(* Logix 5000 project; controller QA_DC vendor 1 type 14 code 164 rev 32.16; software revision 32.04; part 3 of 3 *)
(* tags used below, declared in another part *)
   LN99_1st_Station_Break_Code : DINT;
   LN99_Break_LineWide : BOOL;
   LN99_FROM_DC1_MAIN_MESSAGES : DINT[20];
   LN99_Schedule : UDT_Current_Status;
   LN99_TO_DC1_MAIN_MESSAGE_D : DINT[10];   // WORK CENTER D CONSUME TAG
   LN99_TO_DC1_MAIN_MESSAGE_E : DINT[10];   // WORK CENTER E CONSUME TAG
   LN99_TO_DC1_SUB_MESSAGE_C : DINT[10];   // WORK CENTER C CONSUME TAG
   LN99_TO_DC1_SUB_MESSAGE_E : DINT[10];   // WORK CENTER E CONSUME TAG
   LN99ECS01 : DINT;   // WORK STATION EAST SIDE WORKCENTER C SUBLINE STATION 01
   LN99ECS02 : DINT;   // WORK STATION EAST SIDE WORKCENTER C SUBLINE STATION 02
   LN99ECS03 : DINT;   // WORK STATION EAST SIDE WORKCENTER C SUBLINE STATION 03
   LN99EES01 : DINT;   // WORK STATION EAST SIDE WORK CENTER E SUBLINE STATION 01
   LN99EES02 : DINT;   // WORK STATION EAST SIDE WORK CENTER E SUBLINE STATION 02
   LN99EES03 : DINT;   // WORK STATION EAST SIDE WORK CENTER E SUBLINE STATION 03
   LN99NDM01 : DINT;   // WORK STATION NORTH SIDE WORKCENTER D MAINLINE STATION 01
   LN99NDM02 : DINT;   // WORK STATION NORTH SIDE WORK CENTER D MAINLINE STATION 02
   LN99NDM03 : DINT;   // WORK STATION NORTH SIDE WORK CENTER D MAINLINE STATION 03
   LN99NDM04 : DINT;   // WORK STATION NORTH SIDE WORK CENTER D MAINLINE STATION 04
   LN99NEM01 : DINT;   // WORK STATION NORTH SIDE WORK CENTER E MAIN LINE STATION 01
   LN99NEM02 : DINT;   // WORK STATION NORTH SIDE WORK CENTER E MAINLINE STATION 02
   LN99NEM03 : DINT;   // WORK STATION NORTH SIDE WORK CENTER E MAINLINE STATION 03
   LN99NEM04 : DINT;   // WORK STATION NORTH SIDE WORK CENTER E MAINLINE STATION 04
   LN99NEM05 : DINT;   // WORK STATION NORTH SIDE WORK CENTER E MAINLINE STATION 05
   LN99SDM01 : DINT;   // WORK STATION SOUTH SIDE WORKCENTER D MAINLINE STATION 01
   LN99SDM02 : DINT;   // WORK STATION SOUTH SIDE WORK CENTER D MAINLINE STATION 02
   LN99SDM03 : DINT;   // WORK STATION SOUTH SIDE WORK CENTER D MAINLINE STATION 03
   LN99SDM04 : DINT;   // WORK STATION SOUTH SIDE WORK CENTER D MAINLINE STATION 04
   LN99SEM01 : DINT;   // WORK STATION SOUTH SIDE WORK CENTER E MAINLINE STATION 01
   LN99SEM02 : DINT;   // WORK STATION SOUTH SIDE WORK CENTER E MAINLINE STATION 02
   LN99SEM04 : DINT;   // WORK STATION SOUTH SIDE WORK CENTER E MAINLINE STATION 04
   LN99SEM05 : DINT;   // WORK STATION SOUTH SIDE WORK CENTER E MAINLINE STATION 05
   LN99WCS01 : DINT;   // WORK STATION WEST SIDE WORKCENTER C SUBLINE STATION 01
   LN99WCS02 : DINT;   // WORK STATION WEST SIDE WORKCENTER C SUBLINE STATION 02
   LN99WCS03 : DINT;   // WORK STATION WEST SIDE WORKCENTER C SUBLINE STATION 03
   LN99WES01 : DINT;   // WORK STATION WEST SIDE WORK CENTER E SUBLINE STATION 01
   LN99WES02 : DINT;   // WORK STATION WEST SIDE WORK CENTER E SUBLINE STATION 02
   LN99WES03 : DINT;   // WORK STATION WEST SIDE WORK CENTER E SUBLINE STATION 03
(* LN99, continued *)

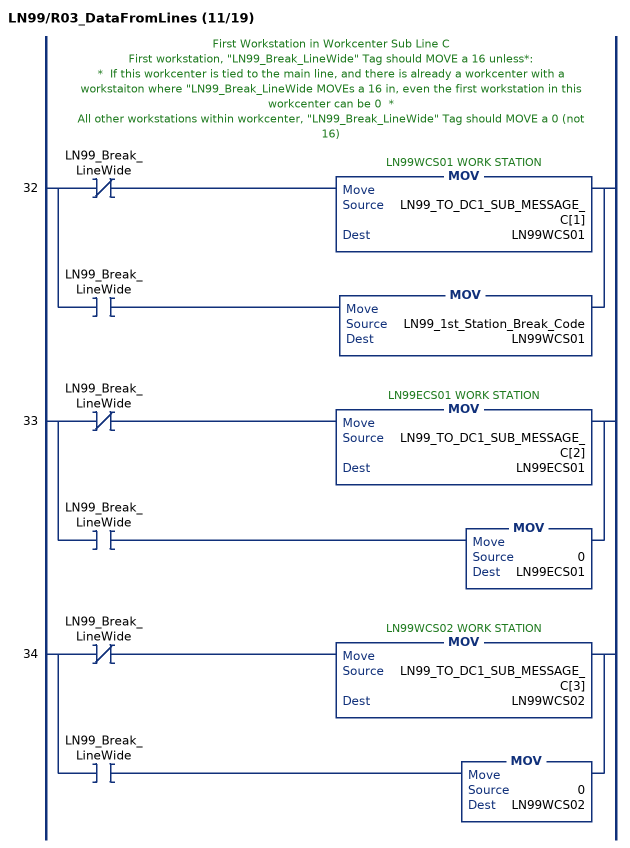
   [picture p52: LN99/R03_DataFromLines rungs 32-34]
   // First Workstation in Workcenter Sub Line C
   // First workstation, "LN99_Break_LineWide" Tag should MOVE a 16 unless*:
   // *  If this workcenter is tied to the main line, and there is already a workcenter with a workstaiton where "LN99_Break_LineWide MOVEs a 16 in, even the first workstation in this workcenter can be 0  *
   // All other workstations within workcenter, "LN99_Break_LineWide" Tag should MOVE a 0 (not 16)
   32: [XIO(LN99_Break_LineWide) MOV(LN99_TO_DC1_SUB_MESSAGE_C[1],LN99WCS01) ,XIC(LN99_Break_LineWide) MOV(LN99_1st_Station_Break_Code,LN99WCS01) ];
   33: [XIO(LN99_Break_LineWide) MOV(LN99_TO_DC1_SUB_MESSAGE_C[2],LN99ECS01) ,XIC(LN99_Break_LineWide) MOV(0,LN99ECS01) ];
   34: [XIO(LN99_Break_LineWide) MOV(LN99_TO_DC1_SUB_MESSAGE_C[3],LN99WCS02) ,XIC(LN99_Break_LineWide) MOV(0,LN99WCS02) ];
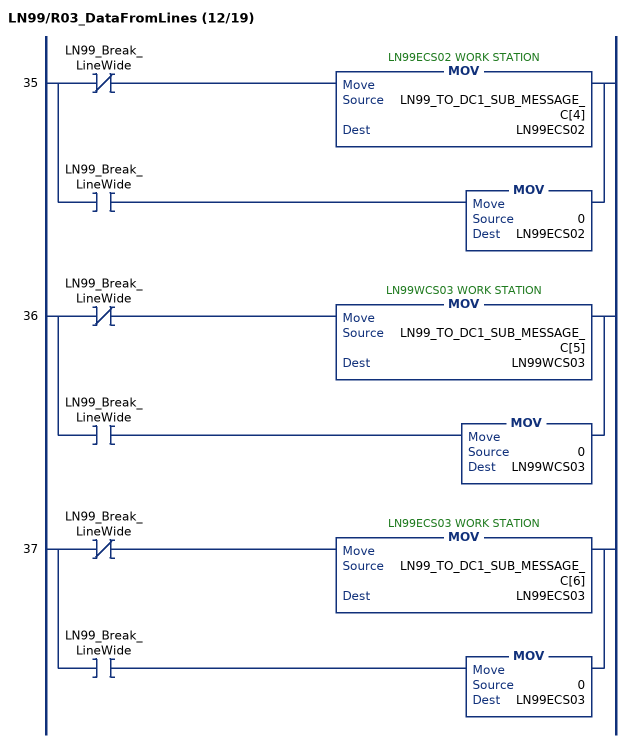
   35: [XIO(LN99_Break_LineWide) MOV(LN99_TO_DC1_SUB_MESSAGE_C[4],LN99ECS02) ,XIC(LN99_Break_LineWide) MOV(0,LN99ECS02) ];
   36: [XIO(LN99_Break_LineWide) MOV(LN99_TO_DC1_SUB_MESSAGE_C[5],LN99WCS03) ,XIC(LN99_Break_LineWide) MOV(0,LN99WCS03) ];
   37: [XIO(LN99_Break_LineWide) MOV(LN99_TO_DC1_SUB_MESSAGE_C[6],LN99ECS03) ,XIC(LN99_Break_LineWide) MOV(0,LN99ECS03) ];
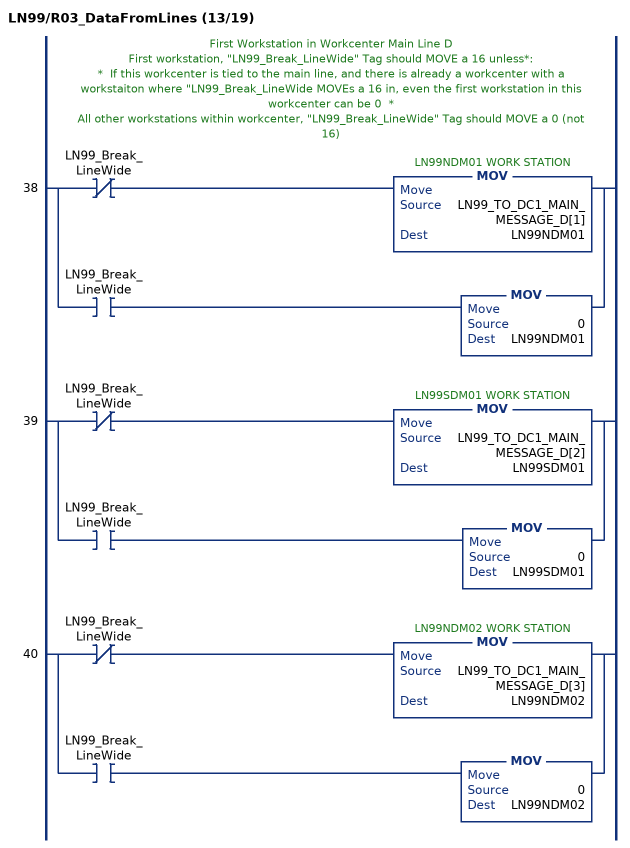
   // First Workstation in Workcenter Main Line D
   // First workstation, "LN99_Break_LineWide" Tag should MOVE a 16 unless*:
   // *  If this workcenter is tied to the main line, and there is already a workcenter with a workstaiton where "LN99_Break_LineWide MOVEs a 16 in, even the first workstation in this workcenter can be 0  *
   // All other workstations within workcenter, "LN99_Break_LineWide" Tag should MOVE a 0 (not 16)
   38: [XIO(LN99_Break_LineWide) MOV(LN99_TO_DC1_MAIN_MESSAGE_D[1],LN99NDM01) ,XIC(LN99_Break_LineWide) MOV(0,LN99NDM01) ];
   39: [XIO(LN99_Break_LineWide) MOV(LN99_TO_DC1_MAIN_MESSAGE_D[2],LN99SDM01) ,XIC(LN99_Break_LineWide) MOV(0,LN99SDM01) ];
   40: [XIO(LN99_Break_LineWide) MOV(LN99_TO_DC1_MAIN_MESSAGE_D[3],LN99NDM02) ,XIC(LN99_Break_LineWide) MOV(0,LN99NDM02) ];
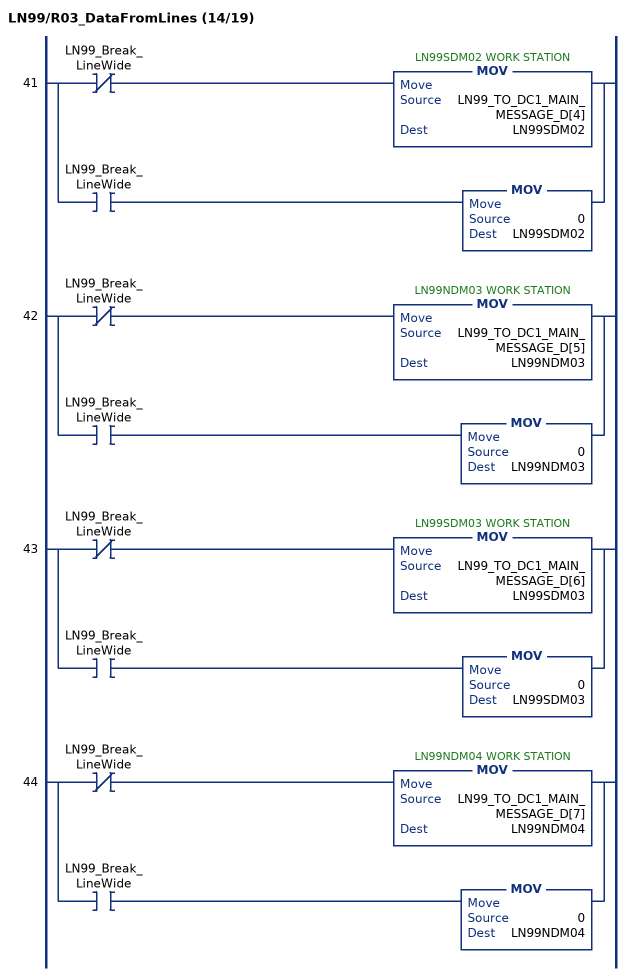
   41: [XIO(LN99_Break_LineWide) MOV(LN99_TO_DC1_MAIN_MESSAGE_D[4],LN99SDM02) ,XIC(LN99_Break_LineWide) MOV(0,LN99SDM02) ];
   42: [XIO(LN99_Break_LineWide) MOV(LN99_TO_DC1_MAIN_MESSAGE_D[5],LN99NDM03) ,XIC(LN99_Break_LineWide) MOV(0,LN99NDM03) ];
   43: [XIO(LN99_Break_LineWide) MOV(LN99_TO_DC1_MAIN_MESSAGE_D[6],LN99SDM03) ,XIC(LN99_Break_LineWide) MOV(0,LN99SDM03) ];
   44: [XIO(LN99_Break_LineWide) MOV(LN99_TO_DC1_MAIN_MESSAGE_D[7],LN99NDM04) ,XIC(LN99_Break_LineWide) MOV(0,LN99NDM04) ];
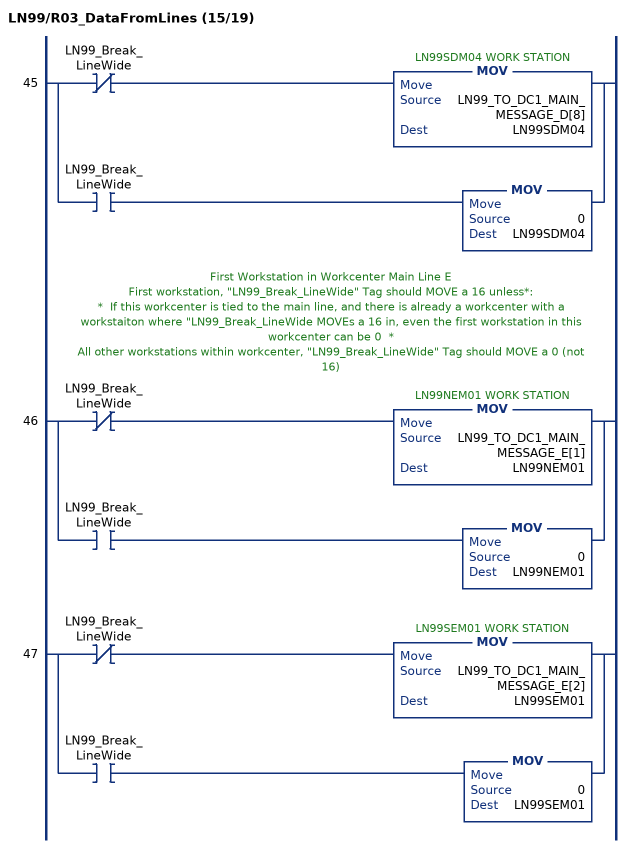
   45: [XIO(LN99_Break_LineWide) MOV(LN99_TO_DC1_MAIN_MESSAGE_D[8],LN99SDM04) ,XIC(LN99_Break_LineWide) MOV(0,LN99SDM04) ];
   // First Workstation in Workcenter Main Line E
   // First workstation, "LN99_Break_LineWide" Tag should MOVE a 16 unless*:
   // *  If this workcenter is tied to the main line, and there is already a workcenter with a workstaiton where "LN99_Break_LineWide MOVEs a 16 in, even the first workstation in this workcenter can be 0  *
   // All other workstations within workcenter, "LN99_Break_LineWide" Tag should MOVE a 0 (not 16)
   46: [XIO(LN99_Break_LineWide) MOV(LN99_TO_DC1_MAIN_MESSAGE_E[1],LN99NEM01) ,XIC(LN99_Break_LineWide) MOV(0,LN99NEM01) ];
   47: [XIO(LN99_Break_LineWide) MOV(LN99_TO_DC1_MAIN_MESSAGE_E[2],LN99SEM01) ,XIC(LN99_Break_LineWide) MOV(0,LN99SEM01) ];
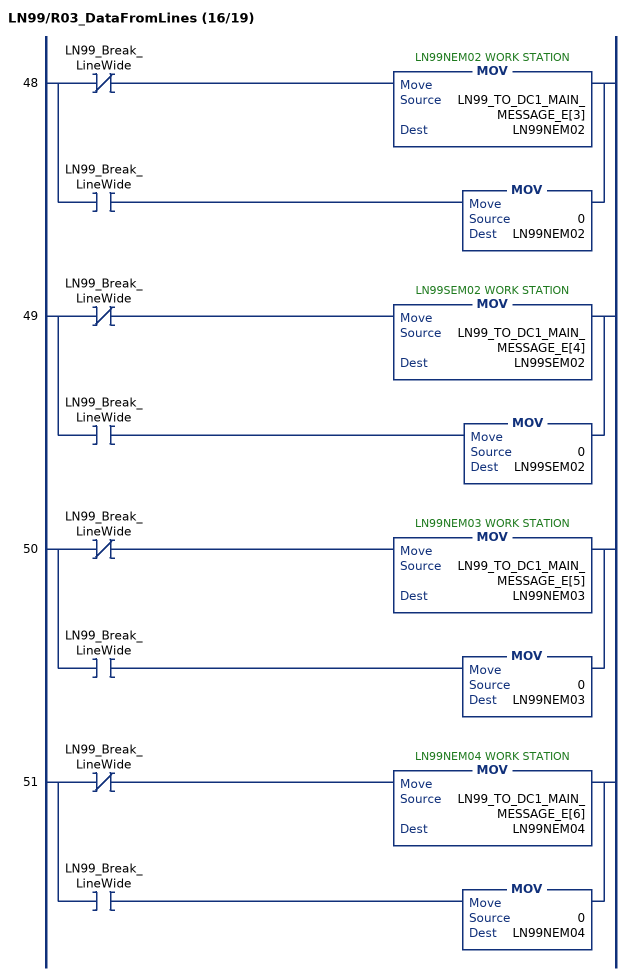
   48: [XIO(LN99_Break_LineWide) MOV(LN99_TO_DC1_MAIN_MESSAGE_E[3],LN99NEM02) ,XIC(LN99_Break_LineWide) MOV(0,LN99NEM02) ];
   49: [XIO(LN99_Break_LineWide) MOV(LN99_TO_DC1_MAIN_MESSAGE_E[4],LN99SEM02) ,XIC(LN99_Break_LineWide) MOV(0,LN99SEM02) ];
   50: [XIO(LN99_Break_LineWide) MOV(LN99_TO_DC1_MAIN_MESSAGE_E[5],LN99NEM03) ,XIC(LN99_Break_LineWide) MOV(0,LN99NEM03) ];
   51: [XIO(LN99_Break_LineWide) MOV(LN99_TO_DC1_MAIN_MESSAGE_E[6],LN99NEM04) ,XIC(LN99_Break_LineWide) MOV(0,LN99NEM04) ];
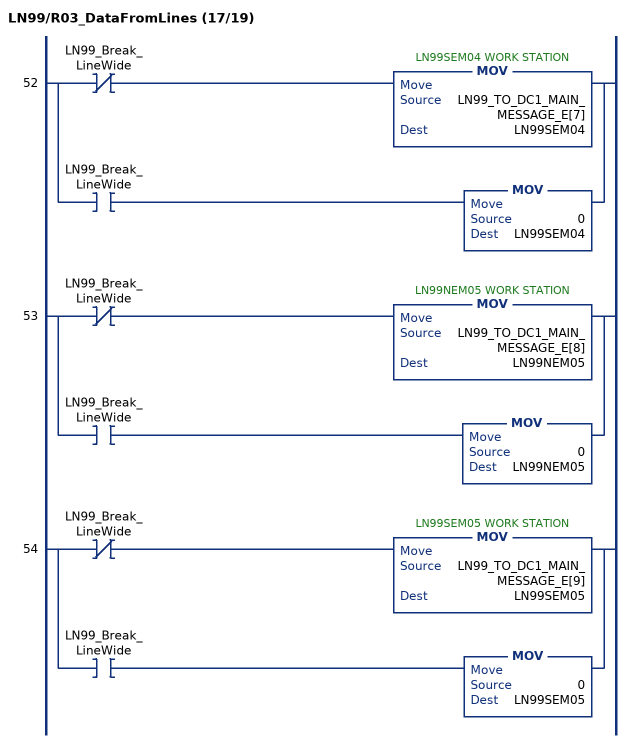
   52: [XIO(LN99_Break_LineWide) MOV(LN99_TO_DC1_MAIN_MESSAGE_E[7],LN99SEM04) ,XIC(LN99_Break_LineWide) MOV(0,LN99SEM04) ];
   53: [XIO(LN99_Break_LineWide) MOV(LN99_TO_DC1_MAIN_MESSAGE_E[8],LN99NEM05) ,XIC(LN99_Break_LineWide) MOV(0,LN99NEM05) ];
   54: [XIO(LN99_Break_LineWide) MOV(LN99_TO_DC1_MAIN_MESSAGE_E[9],LN99SEM05) ,XIC(LN99_Break_LineWide) MOV(0,LN99SEM05) ];
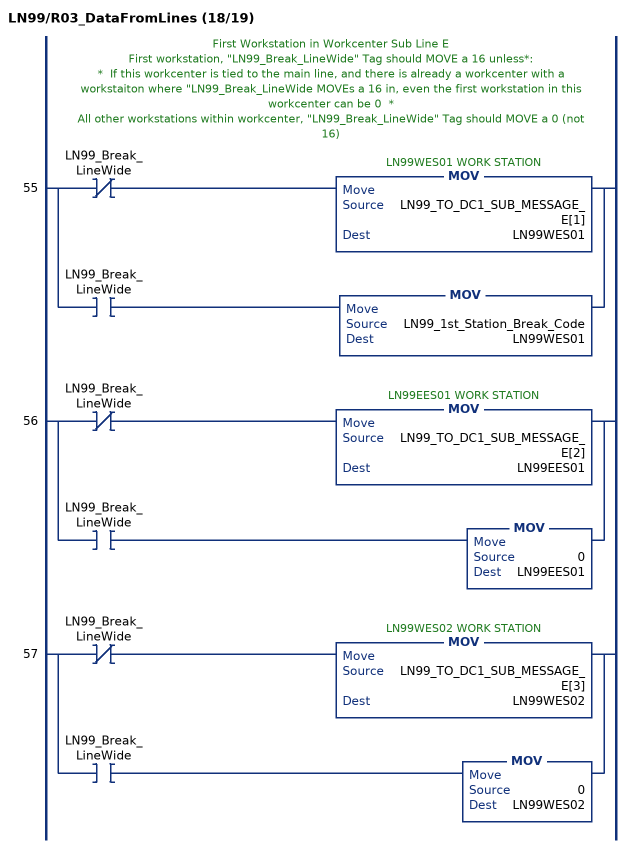
   // First Workstation in Workcenter Sub Line E
   // First workstation, "LN99_Break_LineWide" Tag should MOVE a 16 unless*:
   // *  If this workcenter is tied to the main line, and there is already a workcenter with a workstaiton where "LN99_Break_LineWide MOVEs a 16 in, even the first workstation in this workcenter can be 0  *
   // All other workstations within workcenter, "LN99_Break_LineWide" Tag should MOVE a 0 (not 16)
   55: [XIO(LN99_Break_LineWide) MOV(LN99_TO_DC1_SUB_MESSAGE_E[1],LN99WES01) ,XIC(LN99_Break_LineWide) MOV(LN99_1st_Station_Break_Code,LN99WES01) ];
   56: [XIO(LN99_Break_LineWide) MOV(LN99_TO_DC1_SUB_MESSAGE_E[2],LN99EES01) ,XIC(LN99_Break_LineWide) MOV(0,LN99EES01) ];
   57: [XIO(LN99_Break_LineWide) MOV(LN99_TO_DC1_SUB_MESSAGE_E[3],LN99WES02) ,XIC(LN99_Break_LineWide) MOV(0,LN99WES02) ];
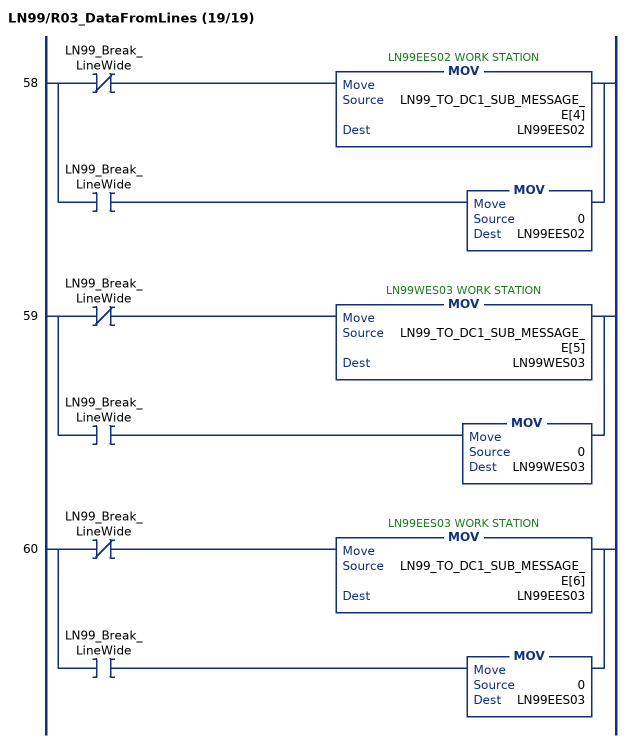
   58: [XIO(LN99_Break_LineWide) MOV(LN99_TO_DC1_SUB_MESSAGE_E[4],LN99EES02) ,XIC(LN99_Break_LineWide) MOV(0,LN99EES02) ];
   59: [XIO(LN99_Break_LineWide) MOV(LN99_TO_DC1_SUB_MESSAGE_E[5],LN99WES03) ,XIC(LN99_Break_LineWide) MOV(0,LN99WES03) ];
   60: [XIO(LN99_Break_LineWide) MOV(LN99_TO_DC1_SUB_MESSAGE_E[6],LN99EES03) ,XIC(LN99_Break_LineWide) MOV(0,LN99EES03) ];
END_ROUTINE

ROUTINE R04_DataToLines   (* ladder *)
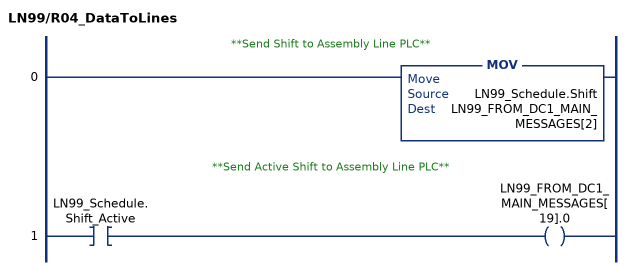
   // **Send Shift to Assembly Line PLC**
   0: MOV(LN99_Schedule.Shift,LN99_FROM_DC1_MAIN_MESSAGES[2]);
   // **Send Active Shift to Assembly Line PLC**
   1: XIC(LN99_Schedule.Shift_Active)OTE(LN99_FROM_DC1_MAIN_MESSAGES[19].0);
END_ROUTINE
END_PROGRAM

PROGRAM MainProgram   (* main routine MainRoutine *)

ROUTINE MainRoutine   (* ladder *)
END_ROUTINE
END_PROGRAM
